// SIMATIC S7-200 project (STEP 7-Micro/WIN), CPU 224XP REL 02.01

SYMBOL_TABLE USUARIO1
marcha_1         I0.0     // enciende e1 y e2
marcha_2         I0.1     // enciende e1
marcha_3         I0.2     // enciende e2
E1               Q0.0     // lampara e1
E2               Q0.1     // lampara e2
L1               M0.0
L2               M0.1
L1_1             M0.2
L2_1             M0.3
PARO             I0.3     // DESCONEXION
END_SYMBOL_TABLE

ORGANIZATION_BLOCK PRINCIPAL:OB1
TITLE=COMENTARIOS DEL PROGRAMA
BEGIN
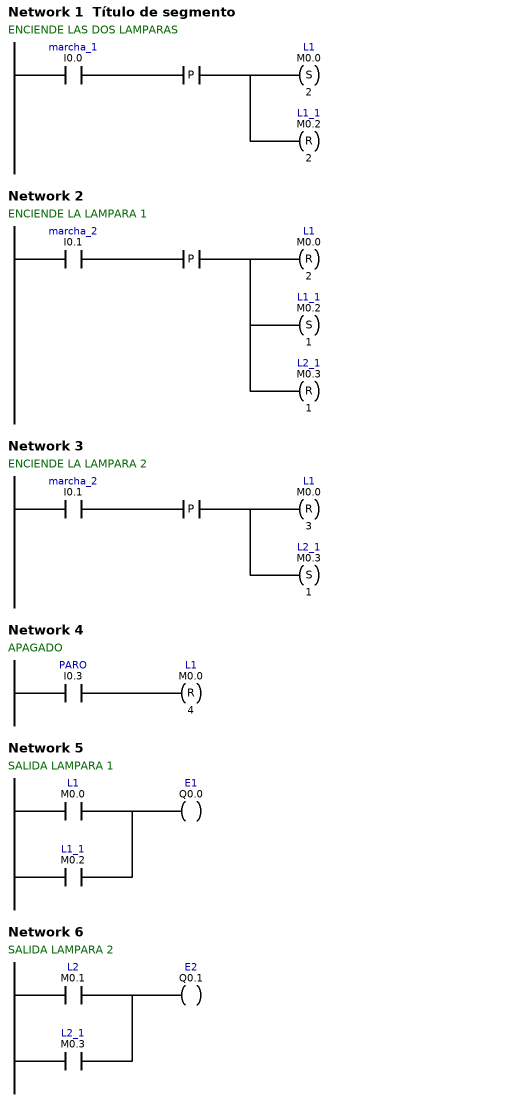
Network 1 // Título de segmento
// ENCIENDE LAS DOS LAMPARAS
LD     marcha_1:I0.0
EU
S      L1:M0.0, 2
R      L1_1:M0.2, 2
Network 2
// ENCIENDE LA LAMPARA 1
LD     marcha_2:I0.1
EU
R      L1:M0.0, 2
S      L1_1:M0.2, 1
R      L2_1:M0.3, 1
Network 3
// ENCIENDE LA LAMPARA 2
LD     marcha_2:I0.1
EU
R      L1:M0.0, 3
S      L2_1:M0.3, 1
Network 4
// APAGADO
LD     PARO:I0.3
R      L1:M0.0, 4
Network 5
// SALIDA LAMPARA 1
LD     L1:M0.0
O      L1_1:M0.2
=      E1:Q0.0
Network 6
// SALIDA LAMPARA 2
LD     L2:M0.1
O      L2_1:M0.3
=      E2:Q0.1
END_ORGANIZATION_BLOCK
